DATA_BLOCK "OP10_GeneralAnalogDB"
{ S7_Optimized_Access := 'TRUE' }
VERSION : 0.1
NON_RETAIN
   VAR RETAIN
      aDev { S7_SetPoint := 'False'} : Array[1..2] of "ST_GeneralAnalog";
   END_VAR


BEGIN

END_DATA_BLOCK

